PROGRAM _ToolLift
VAR_INPUT
	i_bStart					:BOOL;
END_VAR
VAR
	iStep						:INT;
	bRunning					:BOOL;
	tonCheckPos					:TON;
	tonCheckStep				:TON;
	tonTimeOut					:TON;
END_VAR
VAR_OUTPUT
	q_stCmd						:ST_ProcessCmd;
END_VAR

tonTimeOut(IN:=iStep=100,PT:=T#30S);

tonCheckPos(IN:=IN.bMixerTool_InPos,PT:=T#3S);
tonCHeckStep(IN:=iStep=50,PT:=T#5S);

bRunning:=iStep<>0;


CASE iStep OF
	0:
		IF i_bStart AND IN.bToolPos_Down1 AND IN.bToolPos_Down2 THEN
			iStep:=50;
		END_IF
		
	50:
		IF tonCHeckStep.Q THEN
			IF tonCHeckPos.Q THEN
				iStep:=0;
			ELSE
				iStep:=100;
			END_IF
		END_IF
		
	100:
		q_stCmd.rMixerSpeed:=5;
		q_stCmd.bMixerStart:=TRUE;
		IF IN.bMixerTool_InPos THEN
			iStep:=50;
		END_IF
		
		IF tonTimeOut.Q THEN
			iStep:=0;
		END_IF
		
		IF iStep <> 100 THEN
			q_stCmd.rMixerSpeed:=0;
			q_stCmd.bMixerStart:=FALSE;
		END_IF
		
END_CASE

END_PROGRAM

(* stored: Version 1.1.0.1, ProductVersion 3.1.4024.12
   POU _ToolLift: Id {6efbe20f-b4e4-450d-81e6-9cb6f7206718}, SpecialFunc None *)
